// TIA Portal V16 export
// export: Created 2022-01-12T14:34:27.8851906Z, ExportSetting WithDefaults, DisplayName Totally Integrated Automation Portal, DisplayVersion V16 Update 4, DisplayName TIA Portal Version Control Interface, DisplayVersion V16 Update 2, DisplayName TIA Portal Openness, DisplayVersion V16 Update 4, DisplayName STEP 7 Professional, DisplayVersion V16 Update 4, DisplayName STEP 7 Safety, DisplayVersion V16, DisplayName WinCC Professional, DisplayVersion V16 Update 4
TYPE "typSygnałONOFF"
// stored: IsFailsafeCompliant false
   STRUCT
      nazwaSygnału : String[10] := 'F100AV01';
      procedura : Int;   // procedura 0 - to wyłaczenie/procedura 1 to załączenie
      inStart : Bool;
      outStart : Bool;
      hmiTrybAutoManual : Bool;
      hmiManualStart : Bool;
      hmiStanUrządzenia : Int;
   END_STRUCT;
END_TYPE
